INTERFACE I_PROCESS_MAIN EXTENDS I_GENERAL_OBJECT

METHOD M_BreakPressureDet : BOOL
VAR_INPUT
  stBreakPressureParams:                 ST_RECIPE_BREAK_PRESSURE;
END_VAR
END_METHOD

METHOD M_EnduranceRun : BOOL
VAR_INPUT
  stEnduranceRunParams:                 ST_RECIPE_ENDURANCE_RUN;
END_VAR
END_METHOD

METHOD M_EStop : BOOL
VAR_INPUT
END_VAR
END_METHOD

METHOD M_LeakTest1 : BOOL
VAR_INPUT
  stLeakTest1Params:                 ST_RECIPE_LEAK_TEST1;
END_VAR
END_METHOD

METHOD M_LeakTest2 : BOOL
VAR_INPUT
  stLeakTest2Params:                 ST_RECIPE_LEAK_TEST2;
END_VAR
END_METHOD

METHOD M_Reset : BOOL
VAR_INPUT
END_VAR
END_METHOD

METHOD M_SetReady : BOOL
VAR_INPUT
END_VAR
END_METHOD

METHOD M_Stop : BOOL
END_METHOD

METHOD M_StopEngine : BOOL
VAR_INPUT
END_VAR
END_METHOD

PROPERTY P_ReadyState : BOOL
GET
END_GET
END_PROPERTY

END_INTERFACE

(* stored: Version 1.1.0.1, ProductVersion 3.1.4024.12
   Itf I_PROCESS_MAIN: Id {e52b4bdf-1c6c-4901-ab31-ef0200b445fd}
   Method M_BreakPressureDet: Id {168bebf4-bcca-405a-93a9-c6c338d38a37}
   Method M_EnduranceRun: Id {0c7fd0b6-6df4-4b23-a53a-1862430f6423}
   Method M_EStop: Id {1d9039a6-cd46-43d7-ad00-c472b0c618fb}
   Method M_LeakTest1: Id {3109deb2-7598-497d-9b3e-8a27651681b3}
   Method M_LeakTest2: Id {b18a9a37-ce66-473b-ae0a-7cb7751c0ade}
   Method M_Reset: Id {50dc8cf4-d75b-4ab1-9bd3-c504049ff0ed}
   Method M_SetReady: Id {28c5ff99-1e0a-44c5-a1a7-76c3d921bd26}
   Method M_Stop: Id {4e3c4220-9ffb-4900-a309-ce6a74e62206}
   Method M_StopEngine: Id {2b83be8f-92ff-4c65-8d95-f2c9428499cd}
   Property P_ReadyState: Id {50fdb5df-3fb3-4a15-8f1a-5fca3eb252f8}
   Get Get: Id {b0865d3a-4a7b-4f7f-9a17-99e400528a52} *)
